TYPE ST_LaudaReadCommands_SwVersions :
STRUCT
	ControlSyste							: STRING := 'VERSION_R';
	ProtectionSystem						: STRING := 'VERSION_S';
	RemoteControl							: STRING := 'VERSION_B';
	CoolingSystem							: STRING := 'VERSION_T';
	AnalogInterfaceModule					: STRING := 'VERSION_A';
	RS232_422_Profibus_Profinet				: STRING := 'VERSION_V';
	EtherCAT								: STRING := 'VERSION_Z';
	ContactInterace							: STRING := 'VERSION_D';
	SolenoidValveForCoolingWater			: STRING := 'VERSION_M_0';
	SolenoidValveForAutomaticFillingDevice	: STRING := 'VERSION_M_1';
	SolenoidValveForConstantLevelDevice		: STRING := 'VERSION_M_2';
	SolenoidValve_ShutOffValve1				: STRING := 'VERSION_M_3';
	SolenoidValve_ShutOffValve2				: STRING := 'VERSION_M_4';
	ExternalPT100_interface1				: STRING := 'VERSION_E';
END_STRUCT
END_TYPE

(* stored: Version 1.1.0.1, ProductVersion 3.1.4024.12
   DUT ST_LaudaReadCommands_SwVersions: Id {f71baf45-8e40-487e-b25e-733a6ece9306} *)
